FUNCTION_BLOCK FB_GroupTorqueTrimControl_V2
VAR_INPUT
    //----------------------------------------------------------------------
    // TORQUE FEEDBACKS (already filtered)
    //----------------------------------------------------------------------
    group1MasterTorqueFeedback     : REAL;  // EN: Master torque feedback [% or Nm]
    group1Slave1TorqueFeedback     : REAL;  // EN: Slave 1 torque feedback [% or Nm]
    group1Slave2TorqueFeedback     : REAL;  // EN: Slave 2 torque feedback [% or Nm]
    group2MasterTorqueFeedback     : REAL;  // EN: Master torque feedback [% or Nm]
    group2Slave1TorqueFeedback     : REAL;  // EN: Slave 1 torque feedback [% or Nm]
    group2Slave2TorqueFeedback     : REAL;  // EN: Slave 2 torque feedback [% or Nm]

    //----------------------------------------------------------------------
    // CONFIGURATION PARAMETERS
    //----------------------------------------------------------------------
    slaveTorqueOffset              : REAL := 0.0;     // EN: Fixed offset between master and slave [%]
    torqueTrimLimit                : REAL := 10.0;    // EN: Max PID trim output [%]
    torqueLimitMinPct              : REAL := -10.0;     // EN: Min torque command limit [%]
    torqueLimitMaxPct              : REAL := 10.0;   // EN: Max torque command limit [%]

	
	upperAndLowerDifMinPct :  REAL :=  0.1;
	upperAndLowerDifMaxPct	: REAL := -0.1;
	   
	
    //----------------------------------------------------------------------
    // PID GAINS
    //----------------------------------------------------------------------
    torqueCtrlKp                   : REAL := 1.0;
    torqueCtrlTn                   : REAL := 8.0;
    torqueCtrlTv                   : REAL := 0.0;

    upperAndLowerPIDCtrlKp                   : REAL := 0.10;
    upperAndLowerPIDCtrlTn                   : REAL := 1.0;
    tupperAndLowerPIDCtrlTv                   : REAL := 0.0;
	
	
	enableUpperLowerSpeedTrim			: BOOL;
	
    //----------------------------------------------------------------------
    // CONTROL FLAGS
    //----------------------------------------------------------------------
    enableTorquePid                : BOOL := TRUE;    // EN: Enables PID control (FALSE = fixed torque)
END_VAR


VAR_OUTPUT
    //----------------------------------------------------------------------
    // TORQUE REFERENCES (%)
    //----------------------------------------------------------------------
    group1Slave1DriveTorqueRefPct  : REAL;
    group1Slave2DriveTorqueRefPct  : REAL;
    group2Slave1DriveTorqueRefPct  : REAL;
    group2Slave2DriveTorqueRefPct  : REAL;

    //----------------------------------------------------------------------
    // INTERNAL PID OUTPUTS (for monitoring)
    //----------------------------------------------------------------------
    trimGroup1                     : REAL;
    trimGroup2                     : REAL;
	
	
	upperAndLowerSpeedTrim	 	: REAL;
	
	
END_VAR


VAR
    //----------------------------------------------------------------------
    // INTERNAL PID CONTROLLERS
    //----------------------------------------------------------------------
    instCTRL_PID_Group1TorqueTrim  : CTRL_PID;
    instCTRL_PID_Group2TorqueTrim  : CTRL_PID;
    instCTRL_PID_UpperAndLowerSpdTrim  : CTRL_PID;

	
    //----------------------------------------------------------------------
    // INTERNAL SIGNALS
    //----------------------------------------------------------------------
    capMasterGroup1                : REAL;
    capMasterGroup2                : REAL;
    baseLimitGroup1                : REAL;
    baseLimitGroup2                : REAL;
    directTorqueGroup1             : REAL;
    directTorqueGroup2             : REAL;
    avgTorqueGroup1                : REAL;
    avgTorqueGroup2                : REAL;
	upperAndLowerTorqueDif: REAL;
END_VAR


    instCTRL_PID_Group1TorqueTrim(
        ACT := group1Slave1TorqueFeedback,
        SET := group1MasterTorqueFeedback - slaveTorqueOffset,
        MAN := FALSE,
        M_I := 0.0,
        RST := FALSE,
        KP  := torqueCtrlKp,
        TN  := torqueCtrlTn,
        TV  := torqueCtrlTv,
        LL  := torqueLimitMinPct,                   // Bipolar output
        LH  := torqueLimitMaxPct,
		SUP := 1,
        Y   => group1Slave1DriveTorqueRefPct
    );


	
    instCTRL_PID_Group2TorqueTrim(
        ACT := group2Slave1TorqueFeedback,
        SET := group2MasterTorqueFeedback,
        MAN := FALSE,
        M_I := 0.0,
        RST := FALSE,
        KP  := torqueCtrlKp,
        TN  := torqueCtrlTn,
        TV  := torqueCtrlTv,
        LL  := torqueLimitMinPct,                   // Bipolar output
        LH  := torqueLimitMaxPct,
		SUP := 1,		
        Y   => group2Slave1DriveTorqueRefPct
    );


	IF enableUpperLowerSpeedTrim THEN
		
		instCTRL_PID_UpperAndLowerSpdTrim.LL := upperAndLowerDifMinPct;
		instCTRL_PID_UpperAndLowerSpdTrim.LH := upperAndLowerDifMaxPct;
	
	
	ELSE
		
		instCTRL_PID_UpperAndLowerSpdTrim.LL := 0.0;
		instCTRL_PID_UpperAndLowerSpdTrim.LH := 0.0;	
	
	END_IF
	
	
	
		upperAndLowerTorqueDif := group1MasterTorqueFeedback - group2MasterTorqueFeedback;
	
	    instCTRL_PID_UpperAndLowerSpdTrim(
        ACT := upperAndLowerTorqueDif,
        SET := 0,
        MAN := FALSE,
        M_I := 0.0,
        RST := FALSE,
		SUP := 1,
        KP  := upperAndLowerPIDCtrlKp,
        TN  := upperAndLowerPIDCtrlTn,
        TV  := tupperAndLowerPIDCtrlTv,
//        LL  := upperAndLowerDifMinPct,                   // Bipolar output
//        LH  := upperAndLowerDifMaxPct,
        Y   => upperAndLowerSpeedTrim
    );

END_FUNCTION_BLOCK

(* stored: Version 1.1.0.1, ProductVersion 3.1.4024.15
   POU FB_GroupTorqueTrimControl_V2: Id {83cf7ee3-fad9-49c5-8b61-90e194389cd5}, SpecialFunc None *)
